VAR_GLOBAL
(*ExpansionsVentile werden deklariert*)
		EV :	 		ExpansionsVentil; //Dieses Expansionsventil regelt im Normalbetrieb den Verdampfungsdruck und -temperatur
		EV_rev: 		ExpansionsVentil; //Im Falle einer Strömungsumkehrung wird über dieses Expansionsventil in den Verdampfer außerhalb der KlimaKammer eingespritzt
		
(*Zustände der Kältekreiskomponenten: Verdampfer, Verflüssiger, Kompressor, Expansionsventil*)
		EV_in:			Zustandsgroessen;
		EV_rev_in: 		Zustandsgroessen;
		VD : 			Zustandsgroessen;
		VD_rev: 		Zustandsgroessen;
		KP : 			Zustandsgroessen;
		VF : 			Zustandsgroessen;
		VD_defrost : 	Zustandsgroessen;
		
(*Hier ist der Massenstromsensor deklariert*)
		MSS: 			MassenstromSensor;
		
(*Hier sind die Stellsignale für die Ausgangsklemmen deklariert.*)
		Soll_KP: 						OUTPUT_VAR;
		Soll_VF_Ventilator : 			OUTPUT_VAR;
		Soll_VD_defrost_Ventilator : 	OUTPUT_VAR;
		
(*Hier sind alle Heizelemente deklariert.*)
		Soll_ElektHeizrack1 : 			OUTPUT_VAR;		// regelt ein Packet aus 10 Heizstaebe im Verdampfer
		Soll_ElektHeizrack2 : 			OUTPUT_VAR;	 	// regelt ein Packet aus 10 Heizstaebe im Verdampfer
		//Soll_ElektHeizrack3 : 		OUTPUT_VAR;		// !noch nicht im Verdampfer verbaut!
		//Soll_ElektHeizrack4 : 		OUTPUT_VAR;		// !noch nicht im Verdampfer verbaut!
		//Soll_ElektHeizrack5 : 		OUTPUT_VAR;		// !noch nicht im Verdampfer verbaut!
		Soll_ElektHeizrack_Boden: 		OUTPUT_VAR;  	//liegt in der Wanne des Verdampfers, besteht aus 3 Heizstaeben

(*Hier sind alle Drucksensoren deklariert, die im Kältekreislauf installiert sind.
	Die Positionen (Pos) beziehen sich auf das RI-Fließbild von der Kälteanlage*)
		PT_KP_in: 					DruckSensor;		//Pos 1: PT-Sensor vor Kompressor
		PT_KP_out:					DruckSensor;		//Pos 2: PT-Sensor nach Kompressor
		PT_VF_in:					DruckSensor;		//Pos 2': PT-Sensor vor Verflüssiger bzw. nach Abtau-Verdampfer 
		PT_VF_out:					DruckSensor;		//Pos 3': PT-Sensor nach Verflüssiger bzw. vor Abtau-Verdampfer 
		PT_vor_EV 	: 				DruckSensor;		//Pos 3: PT-Sensor vor dem Expansionsventil IV3
		PT_vor_EV_rev : 			DruckSensor;		//Pos 3: PT-Sensor vor dem Expansionsventil IV4,bei Strömungsumkehrung (reverse)
		PT_VD_in	:				DruckSensor;		//Pos 4 : PT-Sensor vor Verdampfer in der Klimakammer 
		PT_VD_out	:				DruckSensor;		//Pos 1': PT-Sensor nach Verdampfer in der Klimakammer 


(*Hier sind alle Temperatursensoren deklariert, die im Kältekreislauf installiert sind.
	Die Positionen (Pos) beziehen sich auf das RI-Fließbild von der Kälteanlage*)
		Temp_VD_in:					INPUT_VAR; //Pos 4: T-Sensor vor Verdampfer in der Klimakammer 
		Temp_VD_out:				INPUT_VAR; //Pos 1': T-Sensor nach Verdampfer in der Klimakammer	
		Temp_VD_in_rev:	 			INPUT_VAR; //Pos 1A': T-Sensor vor Verdampfer bei Strömungsumkehrung(reverse) 	
		Temp_VD_out_rev:			INPUT_VAR; //Pos 4A: T-Sensor nach Verdampfer bei Strömungsumkehrung(reverse)
		Temp_VD_surface1: 			INPUT_VAR; //T-Sensor auf Wärmeübertrager im Verdampfer in der Klimakammer	
		Temp_VD_surface2: 			INPUT_VAR; //T-Sensor auf Wärmeübertrager im Verdampfer in der Klimakammer	
		Temp_VD_surface3: 			INPUT_VAR; //T-Sensor auf Wärmeübertrager im Verdampfer in der Klimakammer	
		Temp_VD_surface4: 			INPUT_VAR; //T-Sensor auf Wärmeübertrager im Verdampfer in der Klimakammer
		Temp_VD_surface5: 			INPUT_VAR; //T-Sensor auf Wärmeübertrager im Verdampfer in der Klimakammer	
		Temp_VD_surface6: 			INPUT_VAR; //T-Sensor auf Wärmeübertrager im Verdampfer in der Klimakammer	
		Temp_VF_in:					INPUT_VAR; // Pos 2': T-Sensor vor Verflüssiger    
		Temp_VF_out: 				INPUT_VAR; // Pos 3': T-Sensor nach Verflüssiger		
		Temp_VD_defrost_in:			INPUT_VAR; // Pos 3A': T-Sensor vor Verdampfer außerhalb der Klimakammer
		Temp_VD_defrost_out:		INPUT_VAR; // Pos 2A': T-Sensor nach Verdampfer außerhalb der Klimakammer
		Temp_KP_in:					INPUT_VAR; // Pos 1: T-Sensor vor Kompressor, im RI-Schema Position 1
		Temp_KP_out:				INPUT_VAR; // Pos 2: T-Sensor nach Kompressor,im RI-Schema Position 2		
		Temp_vor_EV:				INPUT_VAR; // Pos 3: T-Sensor vor dem Expansionsventil IV3
		Temp_vor_EV_rev:			INPUT_VAR; // Pos 3: T-Sensor vor dem Expansionsventil IV4,bei Strömungsumkehrung (reverse)

		Temp_VD_Surface_gemittelt : REAL;

END_VAR

VAR_GLOBAL PERSISTENT
(*Speicherorte für benötigte Stoffwerte. Persistent Variablen sind auch nach Kompilieren und/ oder 
	Neustarten der SPS noch auf dem Arbeitsspeicher des Host-PC´s vorhanden. Die müssen also nicht
	zwangsweise neu eingelesen oder ermittelt werden *)		
		r134a:	ARRAY[1..200] OF Stoffwerte;
		Enthalpie_r134a : ARRAY[-20..100] OF Enthalpie_r134a;
END_VAR

(* stored: Version 1.1.0.1, ProductVersion 3.1.4019.2
   GVL GVL: Id {c411875a-406b-4962-9769-e54fbe539288} *)
